FUNCTION_BLOCK CanInterface_Transporter
VAR_INPUT
END_VAR
VAR_OUTPUT
END_VAR
VAR
	TxData AT%Q* : ST_CanQueue;
	RxData AT%I* : ST_CanQueue;
END_VAR

END_FUNCTION_BLOCK

(* stored: Version 1.1.0.1
   POU CanInterface_Transporter: Id {c60a47cd-3a50-4e37-b37f-89c661c67906}, SpecialFunc None *)
